FUNCTION_BLOCK QUARTER_TO_STR_MEASURED (* quad-state to String *)
  (* Standard: 61499-2 *)
  (* Version 1.0, 2024-02-23, franz *)
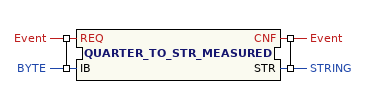
  EVENT_INPUT
    REQ WITH IB; (* Normal Execution Request *)
  END_EVENT
  EVENT_OUTPUT
    CNF WITH STR; (* Execution Confirmation *)
  END_EVENT
  VAR_INPUT
    IB : BYTE := STATUS_DISABLED; (* 2bit (quarter Byte) Output with 4 States *)
  END_VAR
  VAR_OUTPUT
    STR : STRING := STATUS_DISABLED_msg; (* STRING Output *)
  END_VAR
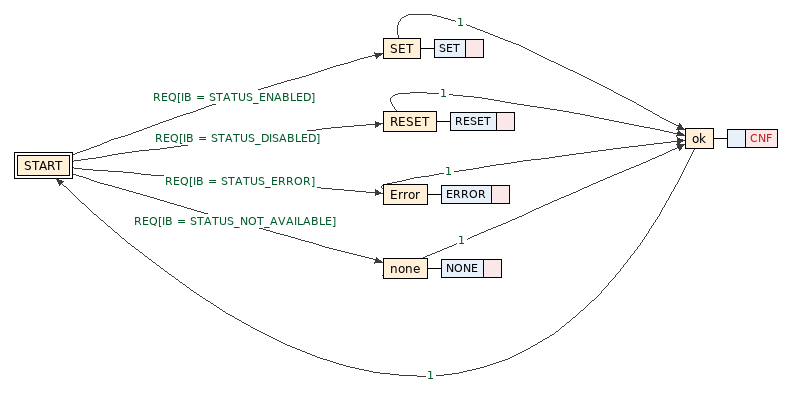
  EC_STATES
    START; (* Initial State *)
    SET : SET;
    RESET : RESET;
    Error : ERROR;
    none : NONE;
    ok : -> CNF;
  END_STATES
  EC_TRANSITIONS
    START TO SET := REQ[IB = STATUS_ENABLED];
    START TO RESET := REQ[IB = STATUS_DISABLED];
    START TO Error := REQ[IB = STATUS_ERROR];
    START TO none := REQ[IB = STATUS_NOT_AVAILABLE];
    SET TO ok := 1;
    RESET TO ok := 1;
    Error TO ok := 1;
    none TO ok := 1;
    ok TO START := 1;
  END_TRANSITIONS
  ALGORITHM SET IN ST:
STR := STATUS_ENABLED_msg;
  END_ALGORITHM
  ALGORITHM RESET IN ST:
STR := STATUS_DISABLED_msg;
  END_ALGORITHM
  ALGORITHM ERROR IN ST:
STR := STATUS_ERROR_msg;
  END_ALGORITHM
  ALGORITHM NONE IN ST:
STR := STATUS_NOT_AVAILABLE_msg;
  END_ALGORITHM
END_FUNCTION_BLOCK
